// TIA Portal V17 export
// export: Created 2024-08-07T21:44:17.6619353Z, ExportSetting WithDefaults, DisplayName Totally Integrated Automation Portal, DisplayVersion V17 Update 7, DisplayName TIA Portal Openness, DisplayVersion V17 Update 7, DisplayName TIA Portal Version Control Interface, DisplayVersion V17, DisplayName SINAMICS Startdrive Advanced, DisplayVersion V17 SP2, DisplayName SINAMICS Startdrive G110M, G120, G120C, G120D, G120P, G115D, DisplayVersion V17 SP2, DisplayName SINAMICS Startdrive G130, G150, S120, S150, SINAMICS MV, S210, DisplayVersion V17 SP2, DisplayName STEP 7 Professional, DisplayVersion V17 Update 7, DisplayName STEP 7 Safety, DisplayVersion V17 Update 6, DisplayName WinCC Advanced / Unified PC, DisplayVersion V17 Update 7
TYPE "typeOpcUaGuid"
// stored: IsFailsafeCompliant false
   STRUCT
      data1 : UDInt;   // Guid values may be represented as a string in this form:<Data1>-<Data2>-<Data3>-<Data4[0:1]>-<Data4[2:7]>
      data2 : UInt;   // A typical Guid value would look like this when formatted as a string: C496578A-0DFE-4b8f-870A-745238C6AEAE
      data3 : UInt;
      data4 : ULInt;
   END_STRUCT;
END_TYPE
